Fanuc KAREL source: kt00367.compact.KL

PROGRAM KT00367
%STACKSIZE=65535
%PRIORITY=65535
%NOLOCKGROUP
VAR
I1 : INTEGER
Y2 : ARRAY[2] OF BYTE
OUT : BOOLEAN
BEGIN
I1=2
Y2[1]=3
OUT=(I1 <=Y2[1])
END KT00367
